// TIA Portal V17 export
// export: Created 2024-08-07T21:44:05.3096758Z, ExportSetting WithDefaults, DisplayName Totally Integrated Automation Portal, DisplayVersion V17 Update 7, DisplayName TIA Portal Openness, DisplayVersion V17 Update 7, DisplayName TIA Portal Version Control Interface, DisplayVersion V17, DisplayName SINAMICS Startdrive Advanced, DisplayVersion V17 SP2, DisplayName SINAMICS Startdrive G110M, G120, G120C, G120D, G120P, G115D, DisplayVersion V17 SP2, DisplayName SINAMICS Startdrive G130, G150, S120, S150, SINAMICS MV, S210, DisplayVersion V17 SP2, DisplayName STEP 7 Professional, DisplayVersion V17 Update 7, DisplayName STEP 7 Safety, DisplayVersion V17 Update 6, DisplayName WinCC Advanced / Unified PC, DisplayVersion V17 Update 7
DATA_BLOCK "Alarms"   // DB20
{ S7_Optimized_Access := 'FALSE' }
VERSION : 0.1
// stored: AutoNumber false, DBAccessibleFromOPCUA true, DBAccessibleFromWebserver true, IsOnlyStoredInLoadMemory false, IsWriteProtectedInAS false
   VAR
      Alarm : Array[1..256] of Bool;
      Warning : Array[1..256] of Bool;
      PartErrorsHMI : Array[1..256] of Bool;
      NOKInAuto : Bool := FALSE;
      Reset : Bool := FALSE;
      ResetHmi : Bool := FALSE;
      AlarmPLC : Array[0..100] of Bool;
   END_VAR
BEGIN
   Alarm[1..256] := FALSE;
   Warning[1..256] := FALSE;
   PartErrorsHMI[1..10] := FALSE;
   PartErrorsHMI[11] := TRUE;
   PartErrorsHMI[12..20] := FALSE;
   PartErrorsHMI[21] := TRUE;
   PartErrorsHMI[22..30] := FALSE;
   PartErrorsHMI[31] := TRUE;
   PartErrorsHMI[32..40] := FALSE;
   PartErrorsHMI[41] := TRUE;
   PartErrorsHMI[42..256] := FALSE;
   AlarmPLC[0..100] := FALSE;
END_DATA_BLOCK
